(* PLC project Generated.project, CODESYS CODESYS V3.5 SP19 Patch 1 *)
(* stored: creationDateTime 2026-09-19T18:18:08.139647, modificationDateTime 2026-09-19T18:18:08.139647 *)

(* ═══════════════════════════════════════════════════════════════ 🕹️ ST_AcquisitionJoystickQualified — Données joystick qualifiées ─────────────────────────────────────────────────────────────── 🎯 Rôle : Encapsuler les commandes d'axes, statut homme-mort et diagnostics produits par FB_Joystick dans PRG_02_Acquisition. 📤 Producteur unique : PRG_02_Acquisition (Data.Joystick). 📄 Doc : DOC/AF/AF_Partie-06_Acquisition_Qualification_IO_v2.4.md ═══════════════════════════════════════════════════════════════ *)
TYPE ST_AcquisitionJoystickQualified : STRUCT
  AxisX : ST_fbJoystick_AxisCmd;  (* 📊 Commande et direction qualifiée axe X *)
  AxisY : ST_fbJoystick_AxisCmd;  (* 📊 Commande et direction qualifiée axe Y *)
  DeadmanArmed : BOOL;  (* 🔒 Homme-mort armé et valide *)
  AtNeutralXY : BOOL;  (* 🟢 Les deux axes X et Y sont au neutre *)
  ArmingPermitDenied : BOOL;  (* ⚠️ Tentative d'armement sans permission *)
  Ready : BOOL;  (* 🟢 Façade joystick prête et opérationnelle *)
  Fault : ST_Fault;  (* ❌ Diagnostic défaut joystick *)
  NeutralXAct : INT;  (* 📍 Valeur ADC neutre calibré X *)
  NeutralYAct : INT;  (* 📍 Valeur ADC neutre calibré Y *)
END_STRUCT;
END_TYPE

(* ======================================================================= ST_Modes_Autorisations - Bus public d'autorisations du mode machine ----------------------------------------------------------------------- Doc metier : DOC/AF/AF_Partie-05_Modes_Maintenance_v2.1.md DOC/AF/AF_Partie-02_Architecture_Programme_v3.2.md #2 NC-110 : le prefixe ST_fb* est reserve aux DUT propriete d'un seul FB. Ce DUT est un BUS multi-consommateurs (>=6 domaines : Cycle, Safety, Treuils, Translation, Supervision, Acquisition) -> renomme ST_Modes_Autorisations (bus de domaine public, sans le prefixe FB). Produit par FB_Modes (via PRG_03_Modes_Cycle) Consomme par : Cycle, Safety, Treuils, Translation, Supervision, Acquisition Producteur unique : FB_Modes (via PRG_03_Modes_Cycle) ======================================================================= *)
TYPE ST_Modes_Autorisations : STRUCT
  Mode : E_Mode;  (* Mode arbitre (DISABLE/N1/N2/SEMI_AUTO) *)
  SyncEnable : BOOL;  (* Synchro M1/M2 (logique positive) *)
  InhibitM1 : BOOL;  (* Inhibition M1 (MAINT_N2 only) *)
  InhibitM2 : BOOL;  (* Inhibition M2 (MAINT_N2 only) *)
  JoystickWinchSelectArbitrated : INT;  (* 0=M1+M2 couples nominal, 1=M1, 2=M2 (unitaires MAINT_N2) *)
  CoupledBucketPhaseLocked : BOOL;  (* T248 : phase mouvement couple VERROUILLEE pour ce maintien joystick -> la perte de l'etat ouvert/ferme en mouvement ne relance PAS de correction benne, ni de blocage "descente/montee interdite". Efface au relachement joystick confirme. *)
  WinchSelTransitionHold : BOOL;  (* T248 : changement de selecteur en cours -> requetes mouvement M1/M2 forcees a 0 jusqu'a l'arret confirme (pas de hand-off en mouvement) *)
  HomingApproachEnable : BOOL;  (* Depassement butee haut (N2) *)
  MaintenanceM3TargetEnable : BOOL;  (* Cible Translation Maintenance (N2 only) *)
  ModeChangePendingBlocked : BOOL;  (* AF-05 #4bis - matrice de maintenance Ces trois champs sont des FAITS/DIAGS publies, pas des autorisations : ils restent vrais meme quand le FB est neutralise par Enable=FALSE (etat persistant). Demande de changement de mode REFUSEE : les treuils *)
  ModeChangeBlockReason : STRING(40);  (* ne sont pas a l'arret mecanique confirme (contacteurs retombes ET frein serre ET |v| < seuil). Mode courant maintenu. Motif du blocage de bascule (texte IHM court, ex. "Chgt mode refuse : contacteur M1") *)
  M1ContactorsReleased : BOOL;  (* Détail des 6 sous-conditions de ModeChangeAllowed (diagnostic IHM) — TRUE = condition satisfaite. M1 : contacteurs retombés *)
  M1BrakeApplied : BOOL;  (* M1 : frein serré (NOT M1BrakeIsOpen) *)
  M1SpeedLow : BOOL;  (* M1 : vitesse sous seuil *)
  M2ContactorsReleased : BOOL;  (* M2 : contacteurs retombés *)
  M2BrakeApplied : BOOL;  (* M2 : frein serré (NOT M2BrakeIsOpen) *)
  M2SpeedLow : BOOL;  (* M2 : vitesse sous seuil *)
  HomingRequiredM1 : BOOL;  (* M1 : re-homing obligatoire avant tout retour SEMI_AUTO *)
  HomingRequiredM2 : BOOL;  (* M2 : idem *)
END_STRUCT;
END_TYPE

(* ======================================================================= 🔌 ST_ProgramWinchRequest — Demande de mouvement treuil par le programme ─────────────────────────────────────────────────────────────── 🎯 Rôle : Regroupe les demandes logiques de treuil formulées par le séquenceur 📄 Référentiel : DOC/WFLOW/CONTRACTS/INTERPRG_CONTRACT_PRG03_MODES_CYCLE_v1.0.md ======================================================================= *)
TYPE ST_ProgramWinchRequest : STRUCT
  RunRequest : BOOL;  (* Ordre marche demandé par le programme *)
  ReqAscent : BOOL;  (* Demande montée *)
  ReqDescend : BOOL;  (* Demande descente *)
  StepTgt : INT;  (* Palier de vitesse cible demandé (1 à 5, 0 = arrêt) *)
END_STRUCT;
END_TYPE

(* ======================================================================= 🎮 ST_WinchBothIntent — Intention both continue de l'opérateur ─────────────────────────────────────────────────────────────── 🎯 Rôle : Transmet l'intention de mouvement both (2 treuils ensemble, homme-mort / boutons) produite inconditionnellement par PRG_03 vers PRG_04 et l'arbitrage (tous modes). Source UNIQUE de la décision both. 📄 Référentiel : DOC/WFLOW/CONTRACTS/INTERPRG_CONTRACT_PRG03_MODES_CYCLE_v1.0.md ======================================================================= *)
TYPE ST_WinchBothIntent : STRUCT
  Active : BOOL;  (* Intention both active (homme-mort qualifié + Select=0 OU boutons BothUp/BothDown) *)
  ReqAscent : BOOL;  (* Intention both montée *)
  ReqDescend : BOOL;  (* Intention both descente *)
END_STRUCT;
END_TYPE

(* ═══════════════════════════════════════════════════════════════ ⚙️ ST_fbWinchCmdArbitration_Cfg — Config treuil (partagé M1/M2) ─────────────────────────────────────────────────────────────── 🎯 Rôle : Config statique de FB_WinchCmdArbitrationM1/M2. Structure UNIQUE partagée : M1 consomme BtnStepTgt (boutons/both), M2 consomme BtnStepTgt (boutons/both) + plafonds benne par sens. 📤 Producteur : PRG_04_Treuils_Benne (câblage). 📄 Doc : DOC/AF/AF_Partie-10_Fonction_Winch_v2.1.md 🔌 Remplace les paliers codés en dur (StepTgt := 5 / StepTgt := 1) par des constantes nommées. ═══════════════════════════════════════════════════════════════ *)
TYPE ST_fbWinchCmdArbitration_Cfg : STRUCT
  BtnStepTgt : INT := 5;  (* --> [CFG] Palier boutons/both (100 % → palier max) *)
  BucketOverrideStepUpTgt : INT := 1;  (* --> [CFG] Plafond benne montée/fermeture *)
  BucketOverrideStepDownTgt : INT := 1;  (* --> [CFG] Plafond benne descente/ouverture *)
  BucketAutoMaxStepUp : INT := 1;  (* --> [CFG] Plafond AX10 fermeture auto (P1..P2, M2 seul) *)
END_STRUCT;
END_TYPE

(* ═══════════════════════════════════════════════════════════════ 🧩 ST_fbWinchCmdArbitration_Context — Contexte de gating treuil (partagé M1/M2) ─────────────────────────────────────────────────────────────── 🎯 Rôle : Encapsuler les faits de gating consommés par FB_WinchCommandArbitrationM1/M2 (benne, synchro, blocage both). Structure UNIQUE partagée par les 2 axes, identifiée par l'instance : M1 ignore le chemin benne, M2 le consomme. 📤 Producteur : PRG_04_Treuils_Benne (câblage). 📄 Doc : DOC/AF/AF_Partie-10_Fonction_Winch_v2.1.md 🔌 Action benne : 2 bits BOOL directionnels M2 issus de FB_Bucket. ═══════════════════════════════════════════════════════════════ *)
TYPE ST_fbWinchCmdArbitration_Context : STRUCT
  BucketBusy : BOOL;  (* --> [STAT] Action benne en cours (instBucket.Lifecycle.Busy) *)
  BucketM2RunRequest : BOOL;  (* --> [CMD] Commande M2 par la benne active *)
  BucketM2ReqAscent : BOOL;  (* --> [CMD] Demande montée M2 issue benne *)
  BucketM2ReqDescend : BOOL;  (* --> [CMD] Demande descente M2 issue benne *)
  BucketAutoCloseActive : BOOL;  (* --> [STAT] AX10 fermeture auto active (plafond AX10 M2, issu de CtrlAscentMaxStep) *)
  BucketHandoffP1Active : BOOL;  (* --> [STAT] AX10B : fermeture atteinte, M2 maintenu au palier 1 avant transfert couple *)
  WinchBothMotionBlockedByBucket : BOOL;  (* --> [STAT] Mouvement both bloqué par benne (ex CoupledMotionBlockedByBucket) *)
  SyncBlocksAscent : BOOL;  (* --> [STAT] Synchro bloque la montée (SyncMinorDeviationBlocksUp) *)
  SyncBlocksDescent : BOOL;  (* --> [STAT] Synchro bloque la descente (SyncMinorDeviationBlocksDown) *)
  M1AscentAllowed : BOOL;  (* === 🔗 ATOMICITÉ DE LA COMMANDE BOTH : permis agrégés consommés === PRG_04 calcule BothAscentPermit/BothDescendPermit = AND des 4 permits effectifs. En commande both, la commande ne consomme QUE ces agrégats (jamais les permits individuels directement) : les 2 treuils partent ensemble ou aucun (NC-100). --> [SAFE] Fait EffectivePermitM1_Ascent *)
  M1DescendAllowed : BOOL;  (* --> [SAFE] Fait EffectivePermitM1_Descend *)
  M2AscentAllowed : BOOL;  (* --> [SAFE] Fait EffectivePermitM2_Ascent *)
  M2DescendAllowed : BOOL;  (* --> [SAFE] Fait EffectivePermitM2_Descend *)
  BothBlock : BOOL;  (* --> [STAT] Commande Both bloquée (aucun départ possible — diagnostic IHM) *)
END_STRUCT;
END_TYPE

(* ═══════════════════════════════════════════════════════════════ 🎛️ ST_fbWinchCmdArbitration_IHM — Entrées IHM de l'arbitrage treuil ─────────────────────────────────────────────────────────────── 🎯 Rôle : Encapsuler les commandes IHM consommées par FB_WinchCommandArbitrationM1/M2 (boutons par treuil, nommage hardware propagé). Le toggle joystick maître global (Modes.Cmd.TglJoystickMaster) est passé en paramètre séparé des FB (I4 — factorisation, source unique GVL_IHM.Modes.Cmd). 📤 Producteur : PRG_04_Treuils_Benne (câblage GVL_IHM). 📄 Doc : DOC/AF/AF_Partie-10_Fonction_Winch_v2.1.md 🔌 Nommage : BtnAscentM1/BtnAscentM2 = nommage hardware propagé (convention projet). ═══════════════════════════════════════════════════════════════ *)
TYPE ST_fbWinchCmdArbitration_IHM : STRUCT
  BtnAscentM1 : BOOL;  (* --> [CMD] Bouton montée treuil M1 (nommage hardware) *)
  BtnDescentM1 : BOOL;  (* --> [CMD] Bouton descente treuil M1 *)
  BtnAscentM2 : BOOL;  (* --> [CMD] Bouton montée treuil M2 *)
  BtnDescentM2 : BOOL;  (* --> [CMD] Bouton descente treuil M2 *)
  BtnWinchBothAscent : BOOL;  (* --> [CMD] Bouton montée couplée both (Commun) *)
  BtnWinchBothDescent : BOOL;  (* --> [CMD] Bouton descente couplée both (Commun) *)
END_STRUCT;
END_TYPE

(* ======================================================================= 🧩 ST_Fault — Brique socle défaut (2 vues : live + latchée) ─────────────────────────────────────────────────────────────── 🎯 Rôle : porter l'état défaut d'un composant, applicable dans TOUS les cas (acquittable ou non), sans brique warning séparée. • Vue LIVE (Error / ErrorId) : suit la cause, retombe seule à 0. • Vue LATCHÉE (Latched / LatchedId): mémorisée au défaut, reste jusqu'au front Reset. Le choix acquittable / non-acquittable se fait PAR CAUSE (ST_FaultCause.Latching), jamais par bloc. 🔒 Sécurité : interlock TOUJOURS sur la cause brute (Error / ErrorId), jamais sur l'acquittement. Reset TOUJOURS effectif, jamais conditionné (std §9). 🧬 Composition : brique de base réutilisable — sortie de FB, struct métier, GVL. Texte IHM NON stocké ici : dérivé côté IHM depuis LatchedId / ErrorId. 📄 Doc : DOC/STDS/CODE_QUALITY_STANDARDS.md §2quinquies / §9 ======================================================================= *)
TYPE ST_Fault : STRUCT
  Error : BOOL;  (* <-- [DIAG] vue LIVE : au moins une cause présente maintenant *)
  ErrorId : WORD;  (* <-- [DIAG] bitfield des causes présentes maintenant (0 si aucune) *)
  Latched : BOOL;  (* <-- [DIAG] vue LATCHÉE : défaut non acquitté, reste jusqu'au front Reset *)
  LatchedId : WORD;  (* <-- [DIAG] ErrorId figé à l'apparition du défaut, effacé au Reset *)
END_STRUCT;
END_TYPE

(* ======================================================================= 🕹️ ST_fbJoystick_AxisCmd — Consigne d'axe normalisée (sortie FB_Joystick) ─────────────────────────────────────────────────────────────── 🎯 Rôle : Structure de consigne d'axe produite par FB_Joystick. 📤 Champs : Enable, StartStop, SpeedTgt (%) + StepTgt (palier 1..5) + direction en bits (DirectionPositive/Negative, AtNeutral). SpeedTgt reste pour l'IHM, StepTgt pour la logique. 📄 Doc métier : DOC/AF/AF_Partie-08_Fonction_Joystick_v2.5.md ======================================================================= *)
TYPE ST_fbJoystick_AxisCmd : STRUCT
  Enable : BOOL;  (* === CONSIGNES DE PILOTAGE AXE === --> [CMD] Autorisation globale pipeline (FALSE=neutralisation, sorties coupees) *)
  StartStop : BOOL;  (* --> [CMD] Validation de mouvement (TRUE=acceleration, FALSE=deceleration/arret) *)
  SpeedTgt : REAL;  (* --> [CMD] Vitesse cible non signee (0...100 %, signe/sens donné par Direction) - IHM *)
  StepTgt : INT;  (* --> [CMD] Palier de vitesse (1..5, 0=arret) - logique/limitations (derive de SpeedTgt) *)
  DirectionNegative : BOOL;  (* --> [CMD] Direction joystick ou intension de gestuelle *)
  DirectionPositive : BOOL;  (* --> [CMD] Direction joystick ou intension de gestuelle *)
  AtNeutral : BOOL;  (* --> [CMD] TRUE si axes en zone morte (position centrale) *)
  Direction : INT;  (* === MONITORING IHM (derive des bits ci-dessus, jamais lu en interlock) === <-- [STAT] Sens -1=Rev / 0=Neutre / +1=Fwd (anim IHM fleche ; lu aussi logique treuils PRG_04) *)
  Deflection : INT;  (* <-- [STAT] Deflexion signee -100..+100 % (anim IHM jauge/barre) *)
END_STRUCT;
END_TYPE

(* values of E_Mode: DISABLE: Mode Désactivé / Veille de sécurité (sorties bloquées); MAINT_N1: Manuel Niveau 1 : Pilotage unitaire avec toutes sécurités actives; MAINT_N2: Manuel Niveau 2 : Pilotage dégradé (droits étendus + bypasses autorisés); SEMI_AUTO: Mode Semi-Automatique (séquenceur automatique) *)

{attribute 'qualified_only'}
{attribute 'strict'}
TYPE E_Mode : (DISABLE := 0, MAINT_N1 := 1, MAINT_N2 := 2, SEMI_AUTO := 3);
END_TYPE

(* ═══════════════════════════════════════════════════════════════ 🪝 FB_WinchCmdArbitrationM2 — Arbitrage de commande treuil M2 ─────────────────────────────────────────────────────────────── 🎯 Rôle : Arbitrer la source de commande M2 (joystick / boutons IHM / demande cycle / chemin benne selon le mode) et produire la commande arbitrée. 🔌 FB d'arbitrage (non-mouvement) : ne porte ni SafeStop ni StartStop de sécurité — il produit la commande logique, la safety reste dans FB_Safety_Winch / FB_Winch. 📄 Doc : DOC/AF/AF_Partie-10_Fonction_Winch_v2.1.md 🔒 Bit-identique à l'ancien PRG_04 §3 (refactor POO). ⚠️ Asymétries M2 vs M1 : chemin benne (override), Select=0/2, synchro inversée. 🪜 -B : la sortie est désormais un PALIER (StepTgt, 1-5) au lieu d'un pourcentage. En SEMI_AUTO, passthrough de ReqWinch.StepTgt ; en manuel, le joystick est le producteur UNIQUE du palier (passthrough de Joystick.AxisY.StepTgt), boutons/both = palier 5, override benne = palier joystick borne par le plafond de configuration. ═══════════════════════════════════════════════════════════════ *)
FUNCTION_BLOCK FB_WinchCmdArbitrationM2
  VAR_INPUT
    Enable : BOOL;  (* --> [CMD] Autorisation FB (TRUE=arbitre actif) *)
    Joystick : ST_AcquisitionJoystickQualified;  (* --> [HW] Données joystick qualifiées (AxisY, DeadmanArmed) *)
    Auth : ST_Modes_Autorisations;  (* --> [CMD] Autorisations mode (Mode, JoystickWinchSelectArbitrated) *)
    ReqWinch : ST_ProgramWinchRequest;  (* --> [REQ] Demande cycle treuil M2 (SEMI_AUTO) *)
    BothIntent : ST_WinchBothIntent;  (* --> [CMD] Intention both opérateur (source unique PRG_03) *)
    IHM : ST_fbWinchCmdArbitration_IHM;  (* --> [CMD] Boutons IHM (BtnAscentM2/BtnDescentM2, both) *)
    TglJoystickMaster : BOOL;  (* --> [CMD] Toggle joystick maître global (Modes.Cmd, source unique) *)
    Context : ST_fbWinchCmdArbitration_Context;  (* --> [STAT] Gating benne/synchro + chemin benne (partagé M1/M2) *)
    Cfg : ST_fbWinchCmdArbitration_Cfg;  (* --> [CFG] Vitesse override benne *)
  END_VAR
  VAR_OUTPUT
    Ready : BOOL;  (* <-- [STAT] FB prêt à arbitrer (Enable) *)
    RunRequest : BOOL;  (* <-- [CMD] Demande marche arbitrée *)
    ReqAscent : BOOL;  (* <-- [CMD] Demande montée arbitrée *)
    ReqDescend : BOOL;  (* <-- [CMD] Demande descente arbitrée *)
    StepTgt : INT;  (* <-- [CMD] Palier de vitesse arbitré (1..5, 0 = arrêt) *)
  END_VAR
  VAR
    BenneBusyFallEdge : F_TRIG;  (* . [LOC] Front descendant action benne (arrêt forcé) *)
    BothDirectionAuthorized : BOOL;  (* . [LOC] Atomicité Both : deux axes autorisés dans le même sens *)
    RequestConflict : BOOL;  (* . [LOC] Double demande de sens refusée *)
    BucketRequestedStep : INT;  (* . [LOC] Palier joystick benne avant plafond de configuration *)
  END_VAR

            

// === IMPLEMENTATION ===

Ready := Enable;

// Front de fin d'action benne (détecté en interne, mécanisme de sécurité)
BenneBusyFallEdge(CLK := Context.BucketBusy);

IF NOT Enable THEN
    RunRequest := FALSE;
    ReqAscent  := FALSE;
    ReqDescend := FALSE;
    StepTgt   := 0;
ELSE
    // ── Chemin benne : M2 piloté par l'action benne (override) ──
    // ⚠️ SÉCURITÉ : l'override benne ne s'applique QUE là où la benne est censée
    // bouger seule (M2 relatif à M1) : jog benne unitaire (WinchSel=2) ou cycle
    // AUTO/SEMI_AUTO qui séquence la benne délibérément. En pilotage COUPLÉ manuel
    // (WinchSel=0) ou unitaire M1 (WinchSel=1), une benne restée Busy NE DOIT PAS
    // détourner M2 : sinon M2 suit la benne pendant que M1 suit le both-intent
    // -> câbles désynchronisés (REX MES 2026-09-04, quasi-casse machine).
    IF Context.BucketBusy AND Context.BucketM2RunRequest
       AND ((Auth.JoystickWinchSelectArbitrated = 2)
            OR (Auth.Mode = E_Mode.SEMI_AUTO)) THEN
        // Axe X translation prioritaire : aucun contacteur treuil pendant un jog X.
        RunRequest := Context.BucketM2RunRequest AND (Joystick.AxisX.Direction = 0);
        ReqAscent  := Context.BucketM2ReqAscent;
        ReqDescend := Context.BucketM2ReqDescend;
        // Le plafond benne borne la consigne joystick ; il ne la remplace pas.
        BucketRequestedStep := LIMIT(1, Joystick.AxisY.StepTgt, 5);
        IF ReqDescend THEN
            StepTgt := MIN(BucketRequestedStep, Cfg.BucketOverrideStepDownTgt);
        ELSIF ReqAscent AND Context.BucketHandoffP1Active THEN
            StepTgt := 1;
        ELSIF ReqAscent AND Context.BucketAutoCloseActive THEN
            StepTgt := MIN(BucketRequestedStep, Cfg.BucketAutoMaxStepUp);
        ELSE
            StepTgt := MIN(BucketRequestedStep, Cfg.BucketOverrideStepUpTgt);
        END_IF;
    ELSE
        // ── Pont SEMI_AUTO : consomme la demande du séquenceur de cycle ──
        IF Auth.Mode = E_Mode.SEMI_AUTO THEN
            // Axe X translation prioritaire : aucun contacteur treuil pendant un jog X.
            RunRequest := ReqWinch.RunRequest AND (Joystick.AxisX.Direction = 0);
            ReqAscent  := ReqWinch.ReqAscent;
            ReqDescend := ReqWinch.ReqDescend;
            StepTgt   := ReqWinch.StepTgt;
        ELSE
            // ── Mode manuel : commande both issue de l'intention UNIQUE PRG_03 (BothIntent),
            //    commande unitaire M2 dérivée des boutons/joystick (Select=2). ──
            // 🪜 StepTgt : le joystick est le producteur UNIQUE du palier (FB_Joystick §6).
            //    Boutons/both = pleine vitesse (100 % → palier 5) ; joystick = passthrough
            //    de Joystick.AxisY.StepTgt. Plus de re-dérivation %→palier ici.
            IF NOT TglJoystickMaster THEN
                // Mode Boutons IHM
                IF BothIntent.Active THEN
                    // Both (BtnWinchBothAscent/Descent) — source unique PRG_03, plus de re-dérivation
                    ReqAscent  := BothIntent.ReqAscent;
                    ReqDescend := BothIntent.ReqDescend;
                    StepTgt   := Cfg.BtnStepTgt;   // 100 % → palier max (configurable)
                ELSIF IHM.BtnAscentM2 THEN
                    ReqAscent  := TRUE;
                    ReqDescend := FALSE;
                    StepTgt   := Cfg.BtnStepTgt;
                ELSIF IHM.BtnDescentM2 THEN
                    ReqAscent  := FALSE;
                    ReqDescend := TRUE;
                    StepTgt   := Cfg.BtnStepTgt;
                ELSE
                    ReqAscent  := FALSE;
                    ReqDescend := FALSE;
                    StepTgt   := 0;
                END_IF;
            ELSE
                // Mode Joystick Maître — M2 unitaire si Select = 2, both si Select = 0
                IF Auth.JoystickWinchSelectArbitrated = 2 THEN
                    ReqAscent  := Joystick.AxisY.Direction > 0;
                    ReqDescend := Joystick.AxisY.Direction < 0;
                    StepTgt   := Joystick.AxisY.StepTgt;
                ELSIF BothIntent.Active THEN
                    // Both (Select=0) — source unique PRG_03, plus de re-dérivation
                    ReqAscent  := BothIntent.ReqAscent;
                    ReqDescend := BothIntent.ReqDescend;
                    StepTgt   := Joystick.AxisY.StepTgt;
                ELSE
                    ReqAscent  := FALSE;
                    ReqDescend := FALSE;
                    StepTgt   := 0;
                END_IF;
            END_IF;

            // Gating StartStop (bit-identique PRG_04 §3) — synchro INVERSÉE vs M1,
            // homme-mort qualifié en joystick
            // 🔗 Atomicité Both : cf. M1 — en both, la commande ne consomme QUE le
            // permit agrégé du sens demandé. Départ jamais isolé entre les 2 treuils.
            RequestConflict := ReqAscent AND ReqDescend;
            BothDirectionAuthorized := (NOT BothIntent.Active)
                OR ((ReqAscent AND NOT ReqDescend) AND Context.M1AscentAllowed AND Context.M2AscentAllowed)
                OR ((ReqDescend AND NOT ReqAscent) AND Context.M1DescendAllowed AND Context.M2DescendAllowed);
            RunRequest := (ReqAscent OR ReqDescend) AND NOT RequestConflict
                      AND NOT Context.WinchBothMotionBlockedByBucket
                      AND NOT ((Context.SyncBlocksAscent   AND ReqDescend)
                            OR (Context.SyncBlocksDescent AND ReqAscent))
                      AND (NOT TglJoystickMaster OR Joystick.DeadmanArmed)
                      // Interlock inter-axes : le jog X translation est prioritaire;
                      // aucun treuil joystick ne part avec X encore deflechi.
                      AND (NOT TglJoystickMaster OR (Joystick.AxisX.Direction = 0))
                      AND BothDirectionAuthorized;
        END_IF;
    END_IF;

    // Front de fin d'action benne : arrêt forcé sauf mouvement both actif
    IF BenneBusyFallEdge.Q AND NOT (BothIntent.Active AND (BothIntent.ReqAscent OR BothIntent.ReqDescend)) THEN
        RunRequest := FALSE;
    END_IF;
END_IF;

          
END_FUNCTION_BLOCK
